FUNCTION_BLOCK Q_GetAttribute (* Command GetAttribute( Part 6 - F.58 ) *)
  (* Standard: ISO 11783-6; Description: This message is available in VT Version 4 and later. This command is used by a Working Set to query the VT for the current state of objects within the VT. Return values iso_s16 - E_NO_ERR - OK - E_OVERFLOW - buffer overflow - E_NOACT - Command not possible in current state - E_NO_INSTANCE - No VT client available *)
  (* Version 1.0, 2022-07-08, franz *)
  (* Documentation:
  This message is available in VT Version 4 and later. This command is used by a Working Set to query the VT for the current state of objects within the VT.
   Return values
   iso_s16
    - E_NO_ERR - OK
   - E_OVERFLOW - buffer overflow
   - E_NOACT - Command not possible in current state
   - E_NO_INSTANCE - No VT client available
  *)
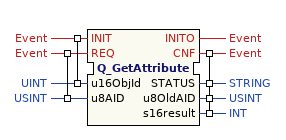
  EVENT_INPUT
    INIT WITH u16ObjId; (* Service Initialization *)
    REQ WITH u8AID; (* Service Request *)
  END_EVENT
  EVENT_OUTPUT
    INITO; (* Initialization Confirm *)
    CNF WITH STATUS, u8OldAID, s16result; (* Confirmation of Requested Service *)
  END_EVENT
  VAR_INPUT
    u16ObjId : UINT; (* Object ID *)
    u8AID : USINT; (* Attribute ID of the object *)
  END_VAR
  VAR_OUTPUT
    STATUS : STRING; (* Service Status *)
    u8OldAID : USINT; (* Old attribute ID of the object *)
    s16result : INT; (* retval see description *)
  END_VAR
END_FUNCTION_BLOCK
